// SIMATIC S7-200 project (STEP 7-Micro/WIN), CPU 224XP CN REL 02.01

ORGANIZATION_BLOCK MAIN:OB1
TITLE=程序注释
BEGIN
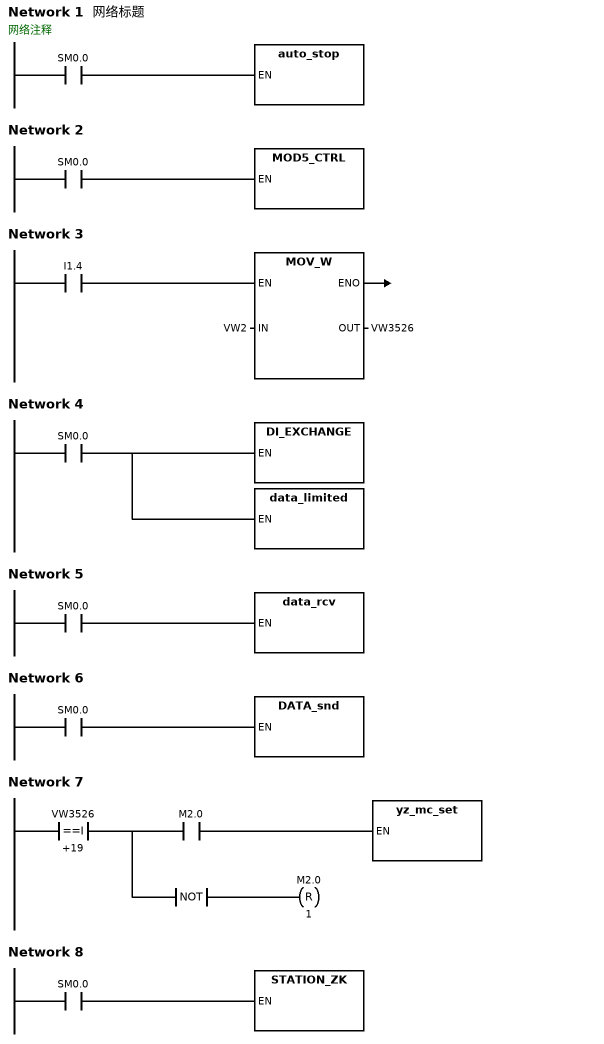
Network 1 // 网络标题
// 网络注释
LD     SM0.0
CALL   auto_stop:SBR13
Network 2
LD     SM0.0
CALL   MOD5_CTRL:SBR12
Network 3
LD     I1.4
MOVW   VW2, VW3526
Network 4
LD     SM0.0
CALL   DI_EXCHANGE:SBR4
CALL   data_limited:SBR9
Network 5
LD     SM0.0
CALL   data_rcv:SBR10
Network 6
LD     SM0.0
CALL   DATA_snd:SBR1
Network 7
LDW=   VW3526, +19
LPS
A      M2.0
CALL   yz_mc_set:SBR6
LPP
NOT
R      M2.0, 1
Network 8
LD     SM0.0
CALL   STATION_ZK:SBR2
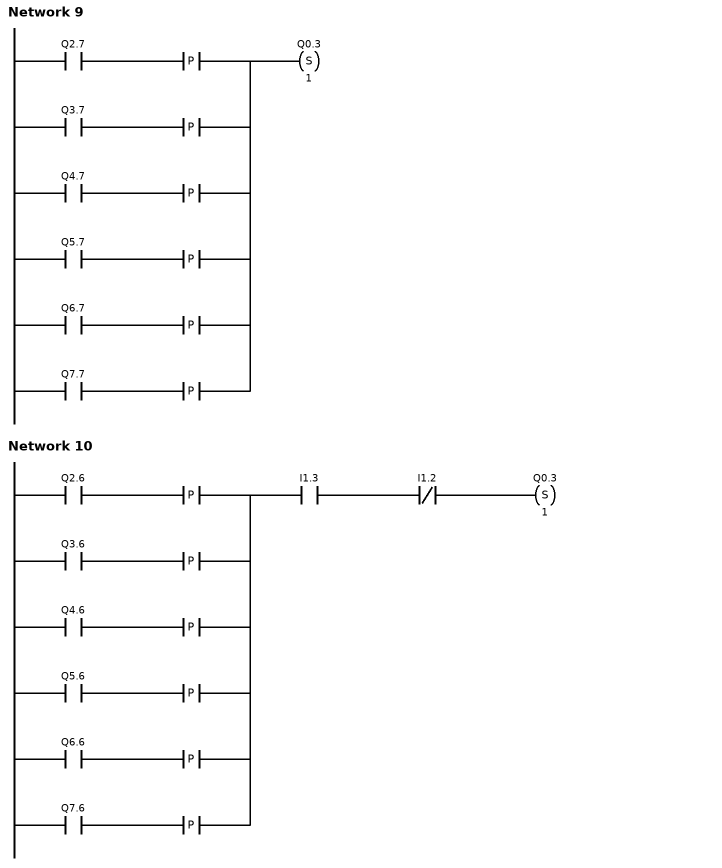
Network 9
LD     Q2.7
EU
LD     Q3.7
EU
OLD
LD     Q4.7
EU
OLD
LD     Q5.7
EU
OLD
LD     Q6.7
EU
OLD
LD     Q7.7
EU
OLD
S      Q0.3, 1
Network 10
LD     Q2.6
EU
LD     Q3.6
EU
OLD
LD     Q4.6
EU
OLD
LD     Q5.6
EU
OLD
LD     Q6.6
EU
OLD
LD     Q7.6
EU
OLD
A      I1.3
AN     I1.2
S      Q0.3, 1
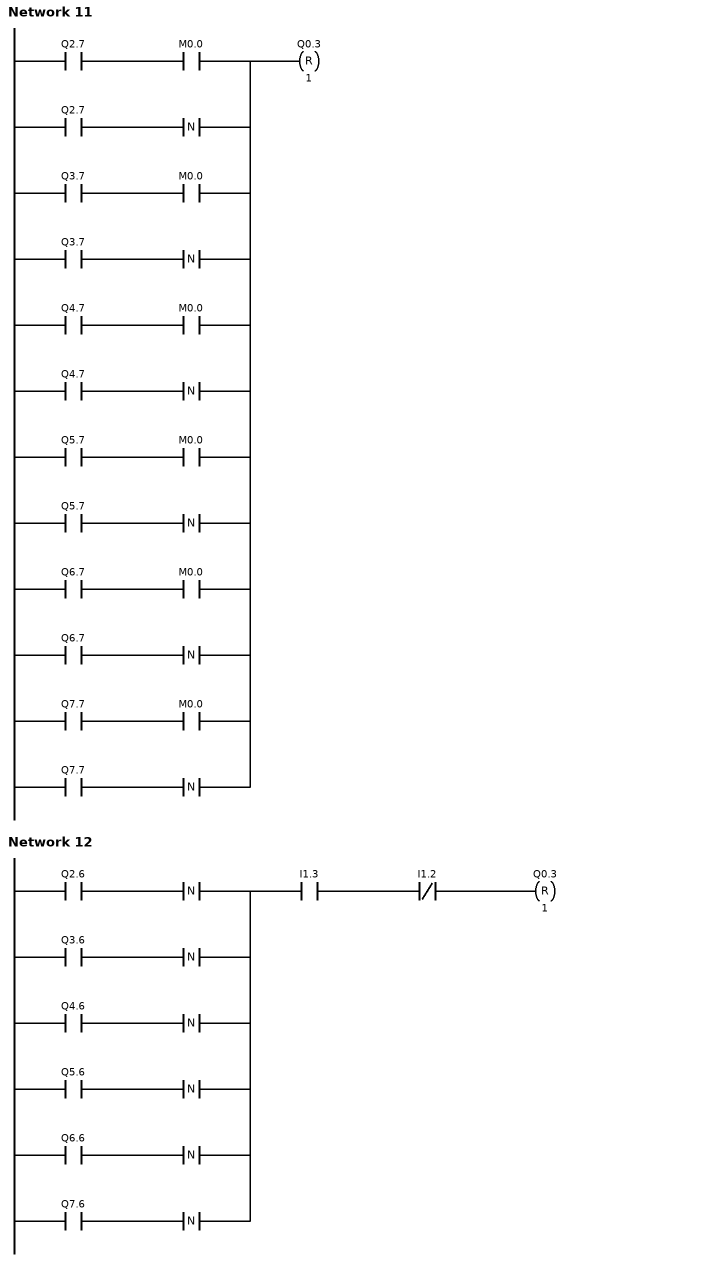
Network 11
LD     Q2.7
A      M0.0
LD     Q2.7
ED
OLD
LD     Q3.7
A      M0.0
OLD
LD     Q3.7
ED
OLD
LD     Q4.7
A      M0.0
OLD
LD     Q4.7
ED
OLD
LD     Q5.7
A      M0.0
OLD
LD     Q5.7
ED
OLD
LD     Q6.7
A      M0.0
OLD
LD     Q6.7
ED
OLD
LD     Q7.7
A      M0.0
OLD
LD     Q7.7
ED
OLD
R      Q0.3, 1
Network 12
LD     Q2.6
ED
LD     Q3.6
ED
OLD
LD     Q4.6
ED
OLD
LD     Q5.6
ED
OLD
LD     Q6.6
ED
OLD
LD     Q7.6
ED
OLD
A      I1.3
AN     I1.2
R      Q0.3, 1
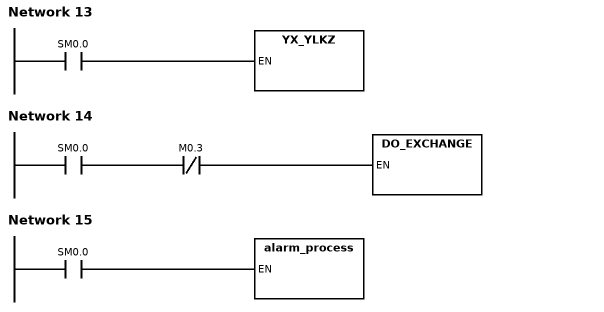
Network 13
LD     SM0.0
CALL   YX_YLKZ:SBR3
Network 14
LD     SM0.0
AN     M0.3
CALL   DO_EXCHANGE:SBR5
Network 15
LD     SM0.0
CALL   alarm_process:SBR11
END_ORGANIZATION_BLOCK

SUBROUTINE_BLOCK STATION_CONTROL:SBR0
TITLE=子程序注释
BEGIN
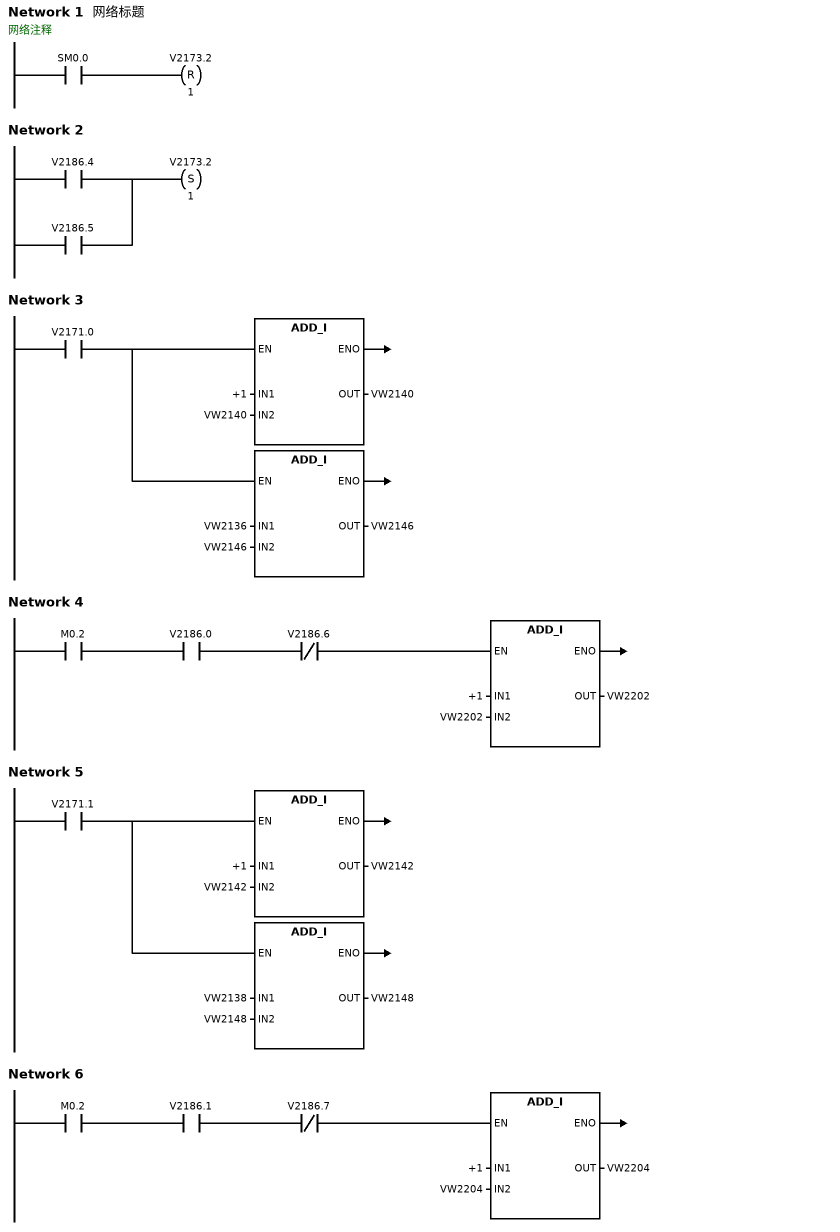
Network 1 // 网络标题
// 网络注释
LD     SM0.0
R      V2173.2, 1
Network 2
LD     V2186.4
O      V2186.5
S      V2173.2, 1
Network 3
LD     V2171.0
+I     +1, VW2140
+I     VW2136, VW2146
Network 4
LD     M0.2
A      V2186.0
AN     V2186.6
+I     +1, VW2202
Network 5
LD     V2171.1
+I     +1, VW2142
+I     VW2138, VW2148
Network 6
LD     M0.2
A      V2186.1
AN     V2186.7
+I     +1, VW2204
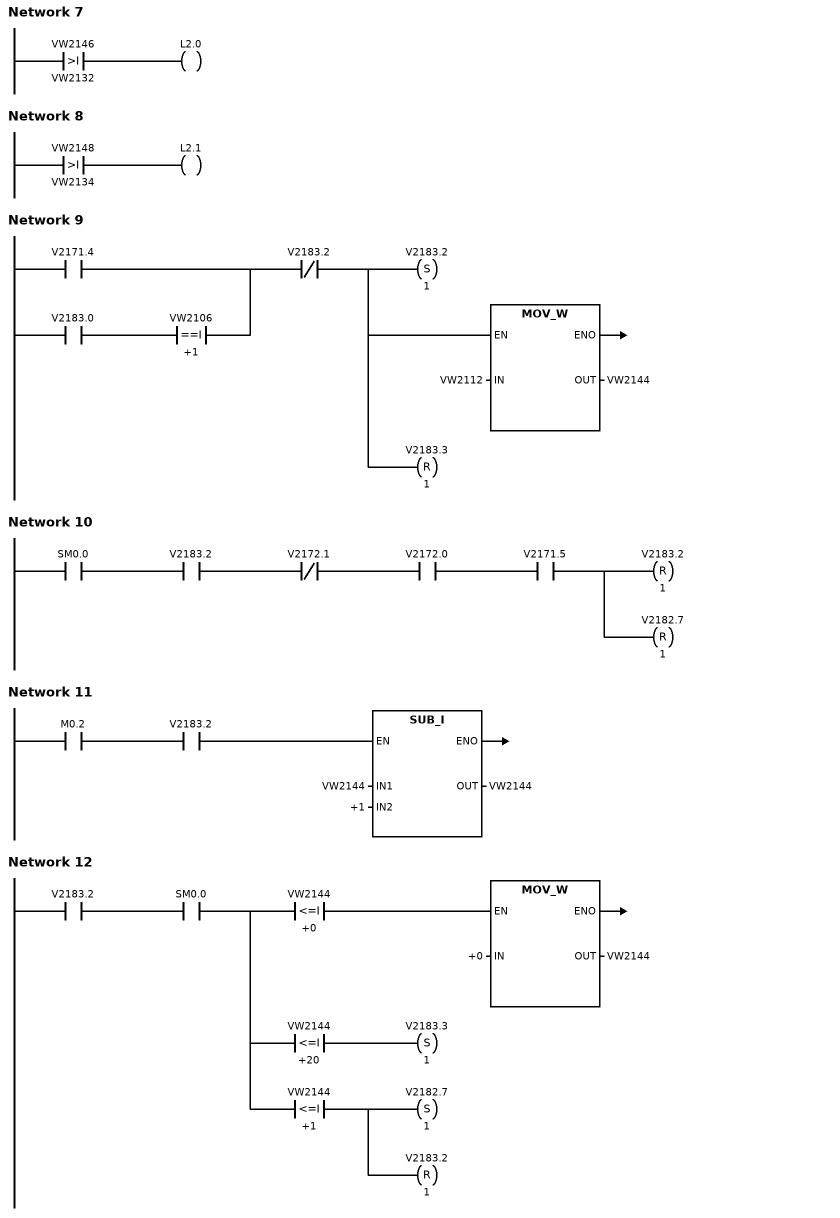
Network 7
LDW>   VW2146, VW2132
=      L2.0
Network 8
LDW>   VW2148, VW2134
=      L2.1
Network 9
LD     V2171.4
LD     V2183.0
AW=    VW2106, +1
OLD
AN     V2183.2
S      V2183.2, 1
MOVW   VW2112, VW2144
R      V2183.3, 1
Network 10
LD     SM0.0
A      V2183.2
AN     V2172.1
A      V2172.0
A      V2171.5
R      V2183.2, 1
R      V2182.7, 1
Network 11
LD     M0.2
A      V2183.2
-I     +1, VW2144
Network 12
LD     V2183.2
A      SM0.0
LPS
AW<=   VW2144, +0
MOVW   +0, VW2144
LRD
AW<=   VW2144, +20
S      V2183.3, 1
LPP
AW<=   VW2144, +1
S      V2182.7, 1
R      V2183.2, 1
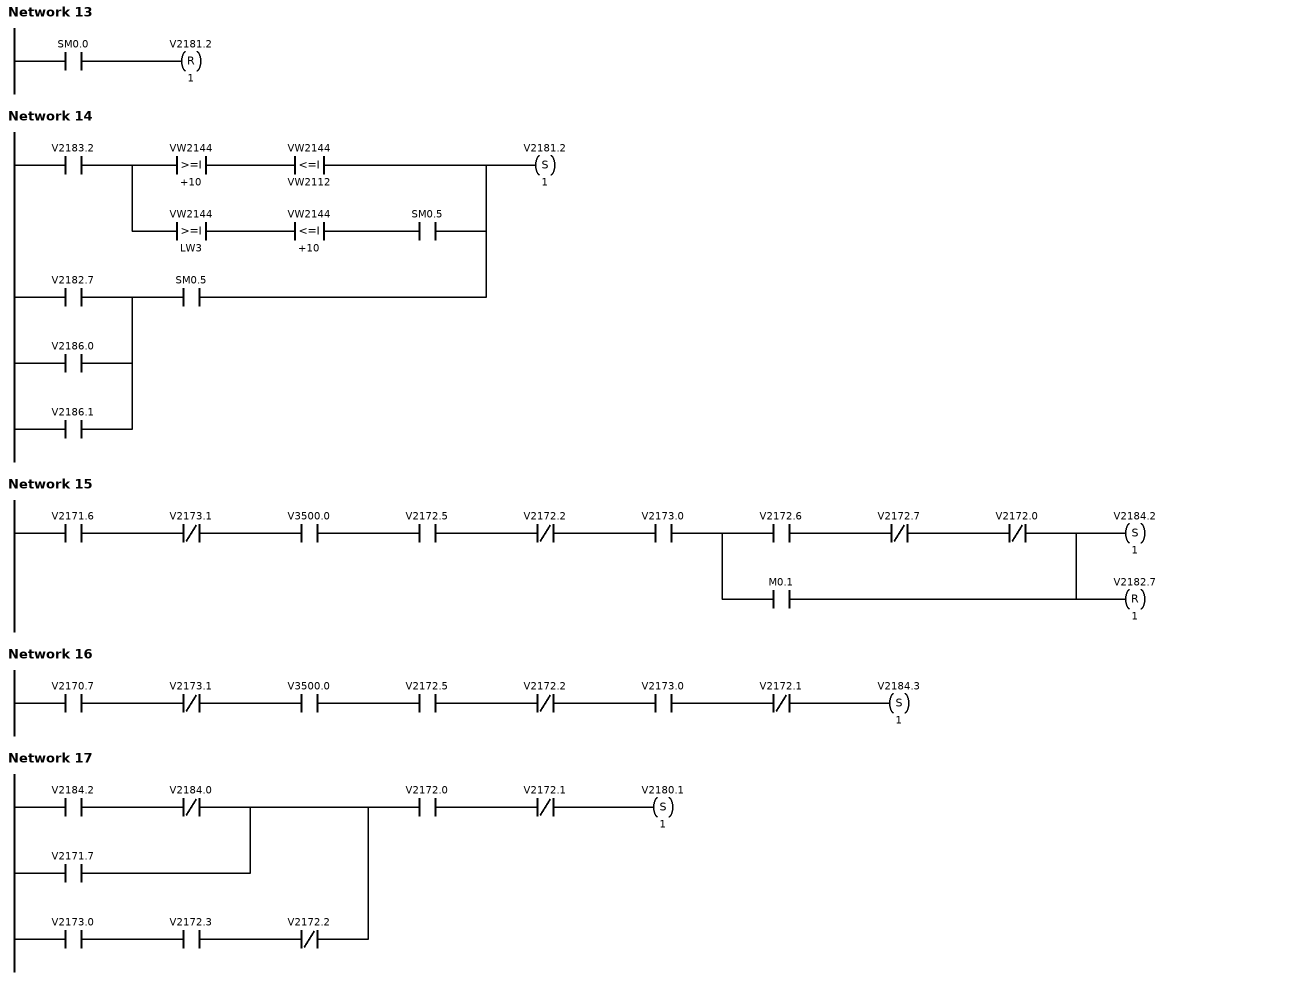
Network 13
LD     SM0.0
R      V2181.2, 1
Network 14
LD     V2183.2
LDW>=  VW2144, +10
AW<=   VW2144, VW2112
LDW>=  VW2144, LW3
AW<=   VW2144, +10
A      SM0.5
OLD
ALD
LD     V2182.7
O      V2186.0
O      V2186.1
A      SM0.5
OLD
S      V2181.2, 1
Network 15
LD     V2171.6
AN     V2173.1
A      V3500.0
A      V2172.5
AN     V2172.2
A      V2173.0
LD     V2172.6
AN     V2172.7
AN     V2172.0
O      M0.1
ALD
S      V2184.2, 1
R      V2182.7, 1
Network 16
LD     V2170.7
AN     V2173.1
A      V3500.0
A      V2172.5
AN     V2172.2
A      V2173.0
AN     V2172.1
S      V2184.3, 1
Network 17
LD     V2184.2
AN     V2184.0
O      V2171.7
LD     V2173.0
A      V2172.3
AN     V2172.2
OLD
A      V2172.0
AN     V2172.1
S      V2180.1, 1
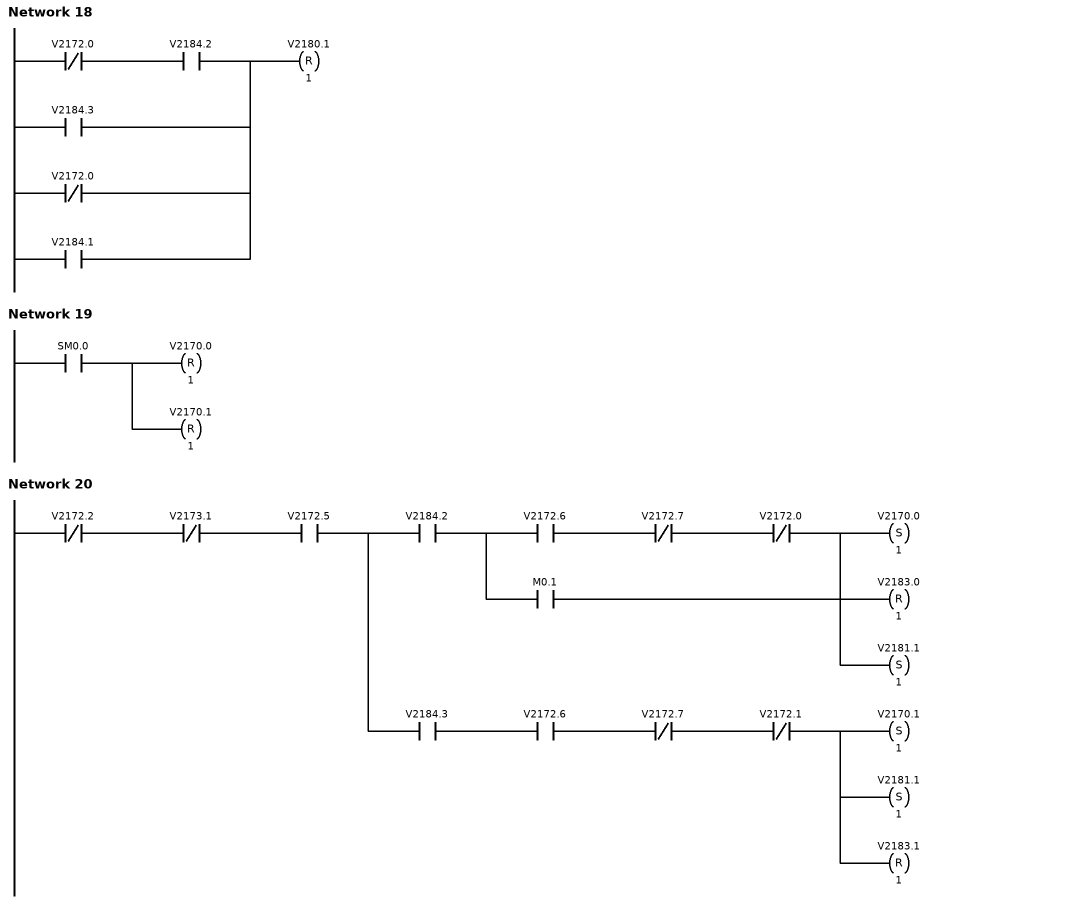
Network 18
LDN    V2172.0
A      V2184.2
O      V2184.3
ON     V2172.0
O      V2184.1
R      V2180.1, 1
Network 19
LD     SM0.0
R      V2170.0, 1
R      V2170.1, 1
Network 20
LDN    V2172.2
AN     V2173.1
A      V2172.5
LPS
A      V2184.2
LD     V2172.6
AN     V2172.7
AN     V2172.0
O      M0.1
ALD
S      V2170.0, 1
R      V2183.0, 1
S      V2181.1, 1
LPP
A      V2184.3
A      V2172.6
AN     V2172.7
AN     V2172.1
S      V2170.1, 1
S      V2181.1, 1
R      V2183.1, 1
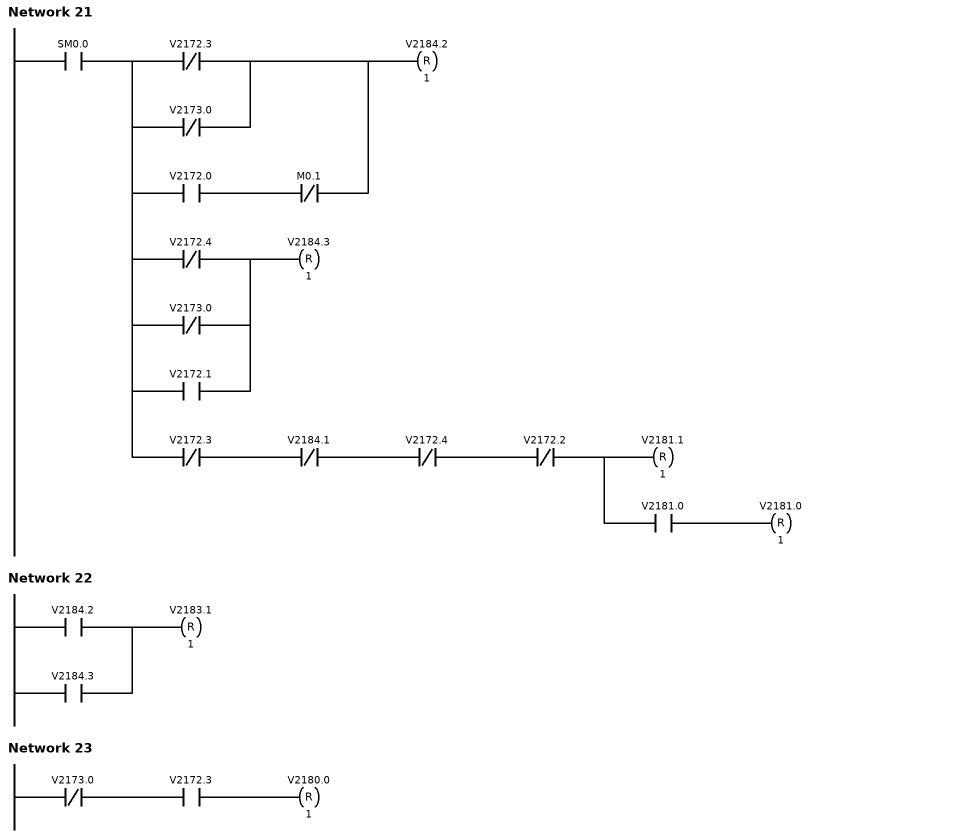
Network 21
LD     SM0.0
LPS
LDN    V2172.3
ON     V2173.0
LD     V2172.0
AN     M0.1
OLD
ALD
R      V2184.2, 1
LRD
LDN    V2172.4
ON     V2173.0
O      V2172.1
ALD
R      V2184.3, 1
LPP
AN     V2172.3
AN     V2184.1
AN     V2172.4
AN     V2172.2
R      V2181.1, 1
A      V2181.0
R      V2181.0, 1
Network 22
LD     V2184.2
O      V2184.3
R      V2183.1, 1
Network 23
LDN    V2173.0
A      V2172.3
R      V2180.0, 1
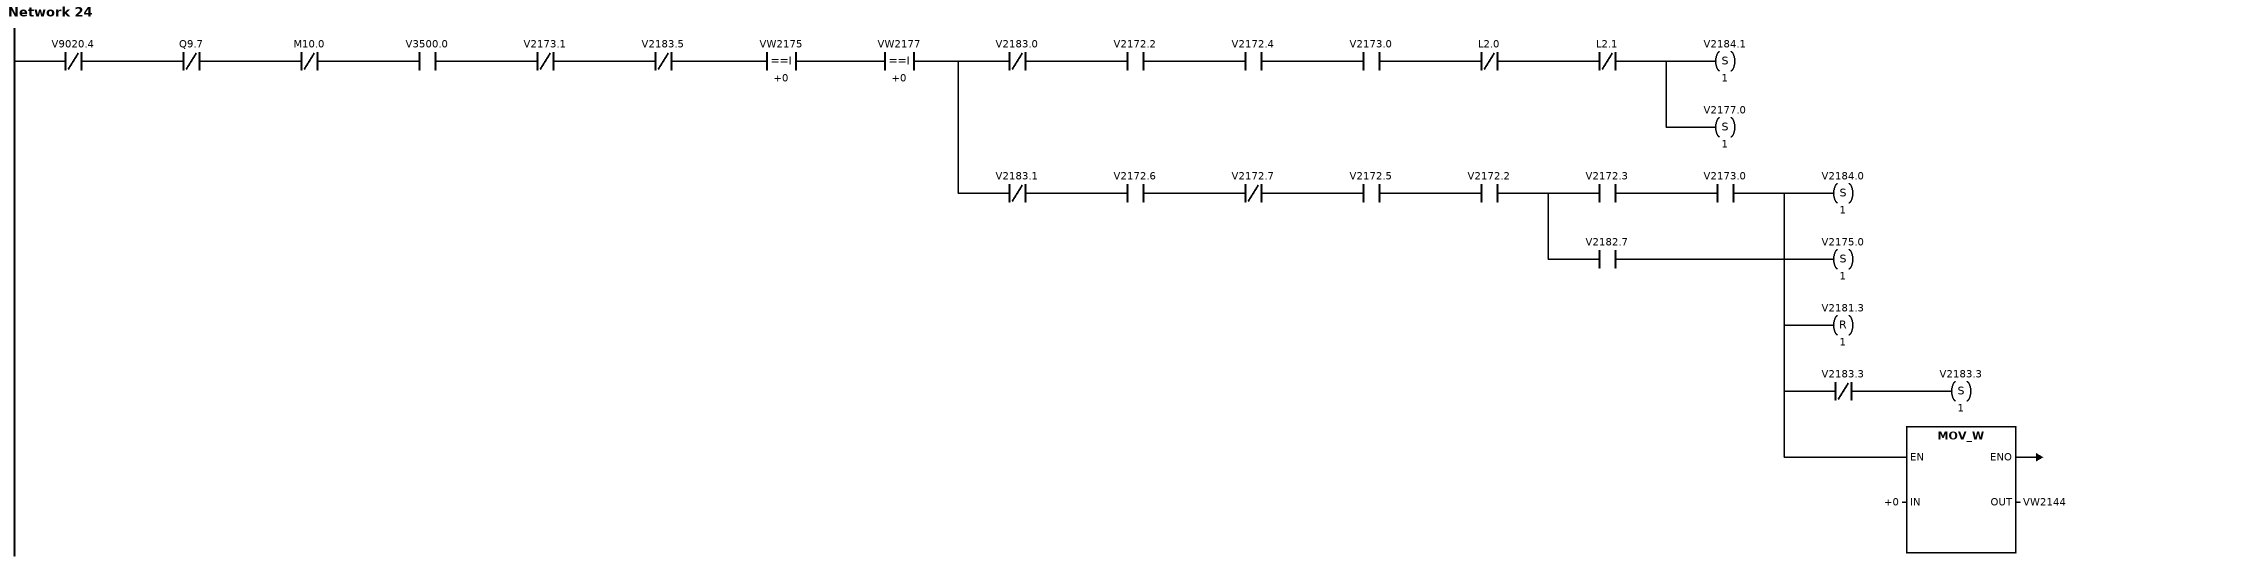
Network 24
LDN    V9020.4
AN     Q9.7
AN     M10.0
A      V3500.0
AN     V2173.1
AN     V2183.5
AW=    VW2175, +0
AW=    VW2177, +0
LPS
AN     V2183.0
A      V2172.2
A      V2172.4
A      V2173.0
AN     L2.0
AN     L2.1
S      V2184.1, 1
S      V2177.0, 1
LPP
AN     V2183.1
A      V2172.6
AN     V2172.7
A      V2172.5
A      V2172.2
LD     V2172.3
A      V2173.0
O      V2182.7
ALD
LPS
S      V2184.0, 1
S      V2175.0, 1
R      V2181.3, 1
AN     V2183.3
S      V2183.3, 1
LPP
MOVW   +0, VW2144
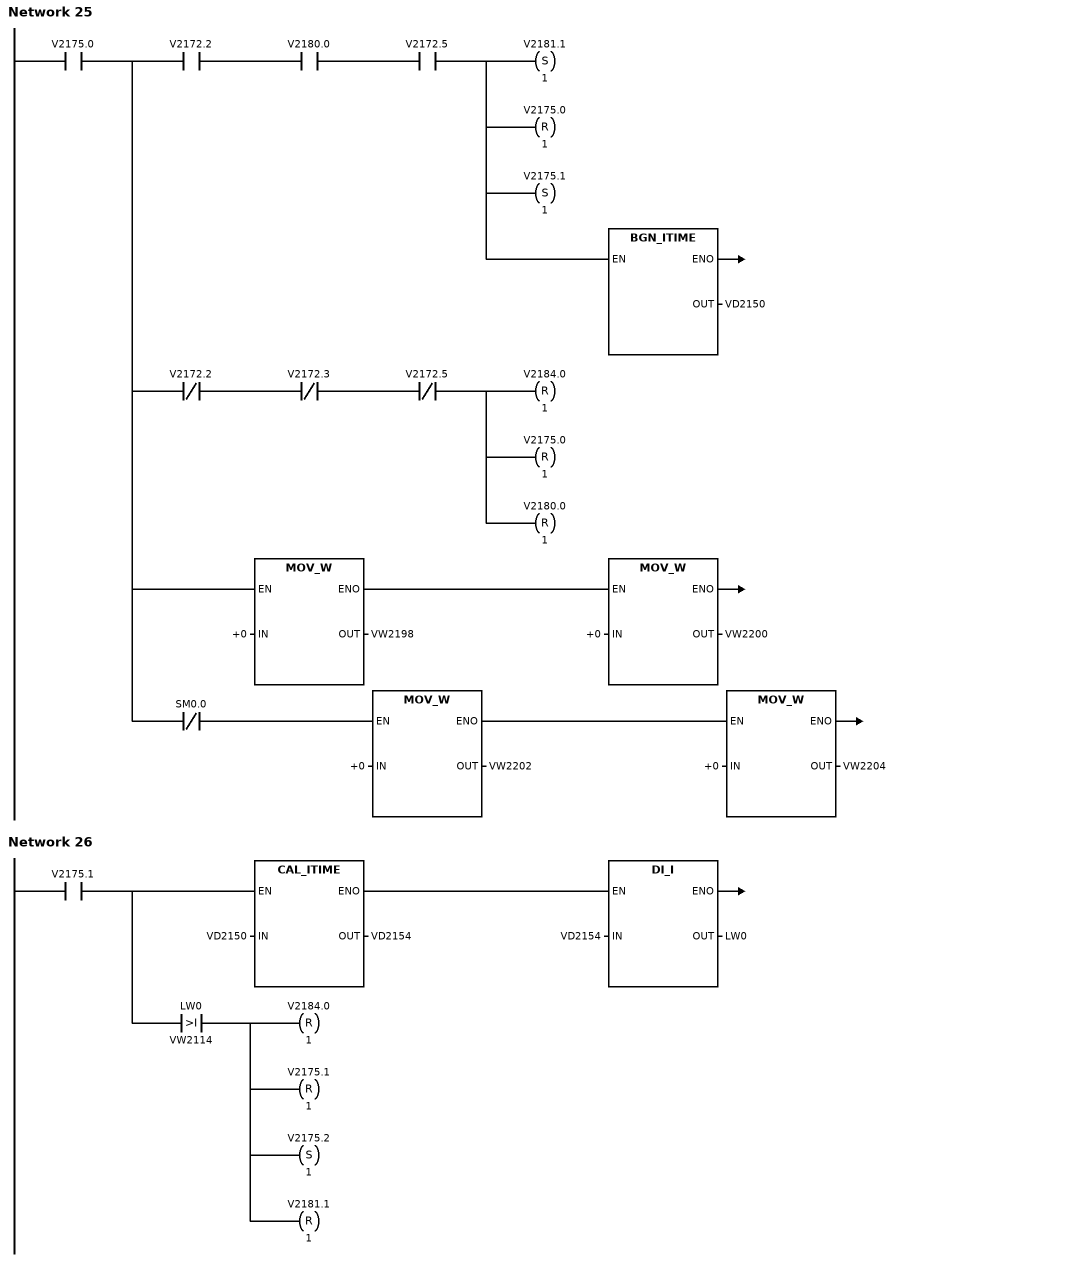
Network 25
LD     V2175.0
LPS
A      V2172.2
A      V2180.0
A      V2172.5
S      V2181.1, 1
R      V2175.0, 1
S      V2175.1, 1
BITIM  VD2150
LRD
AN     V2172.2
AN     V2172.3
AN     V2172.5
R      V2184.0, 1
R      V2175.0, 1
R      V2180.0, 1
LPP
LPS
MOVW   +0, VW2198
AENO
MOVW   +0, VW2200
LPP
AN     SM0.0
MOVW   +0, VW2202
AENO
MOVW   +0, VW2204
Network 26
LD     V2175.1
LPS
CITIM  VD2150, VD2154
AENO
DTI    VD2154, LW0
LPP
AW>    LW0, VW2114
R      V2184.0, 1
R      V2175.1, 1
S      V2175.2, 1
R      V2181.1, 1
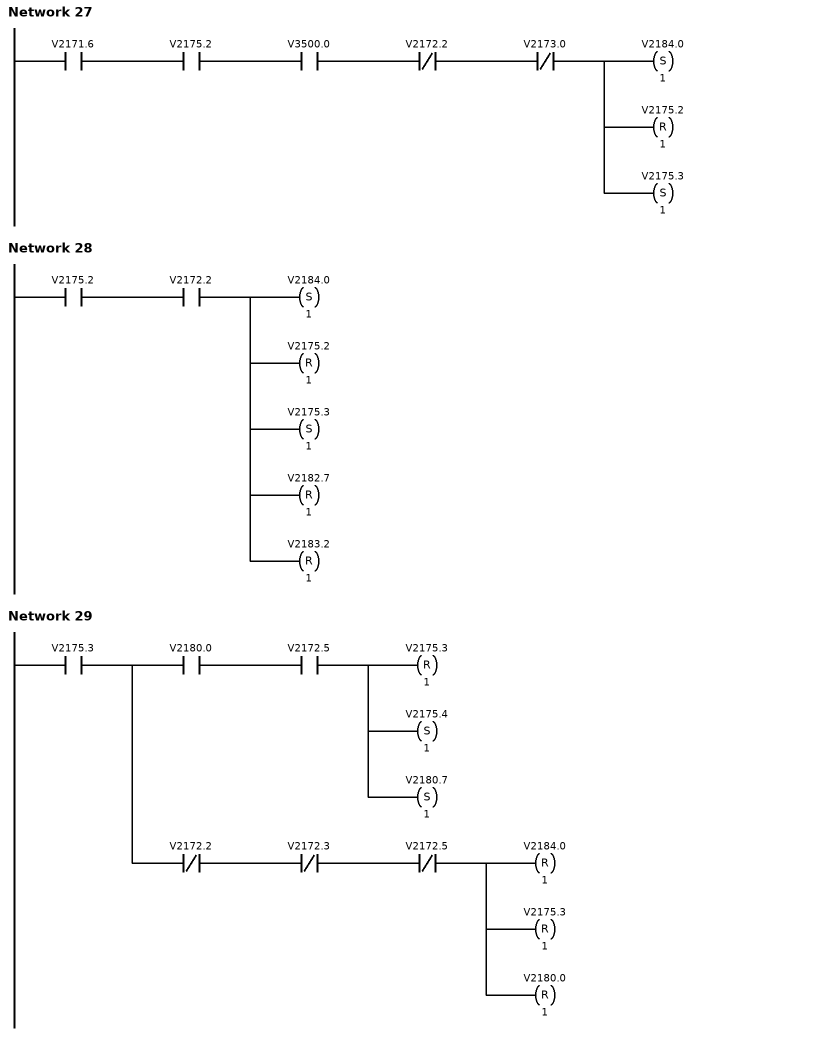
Network 27
LD     V2171.6
A      V2175.2
A      V3500.0
AN     V2172.2
AN     V2173.0
S      V2184.0, 1
R      V2175.2, 1
S      V2175.3, 1
Network 28
LD     V2175.2
A      V2172.2
S      V2184.0, 1
R      V2175.2, 1
S      V2175.3, 1
R      V2182.7, 1
R      V2183.2, 1
Network 29
LD     V2175.3
LPS
A      V2180.0
A      V2172.5
R      V2175.3, 1
S      V2175.4, 1
S      V2180.7, 1
LPP
AN     V2172.2
AN     V2172.3
AN     V2172.5
R      V2184.0, 1
R      V2175.3, 1
R      V2180.0, 1
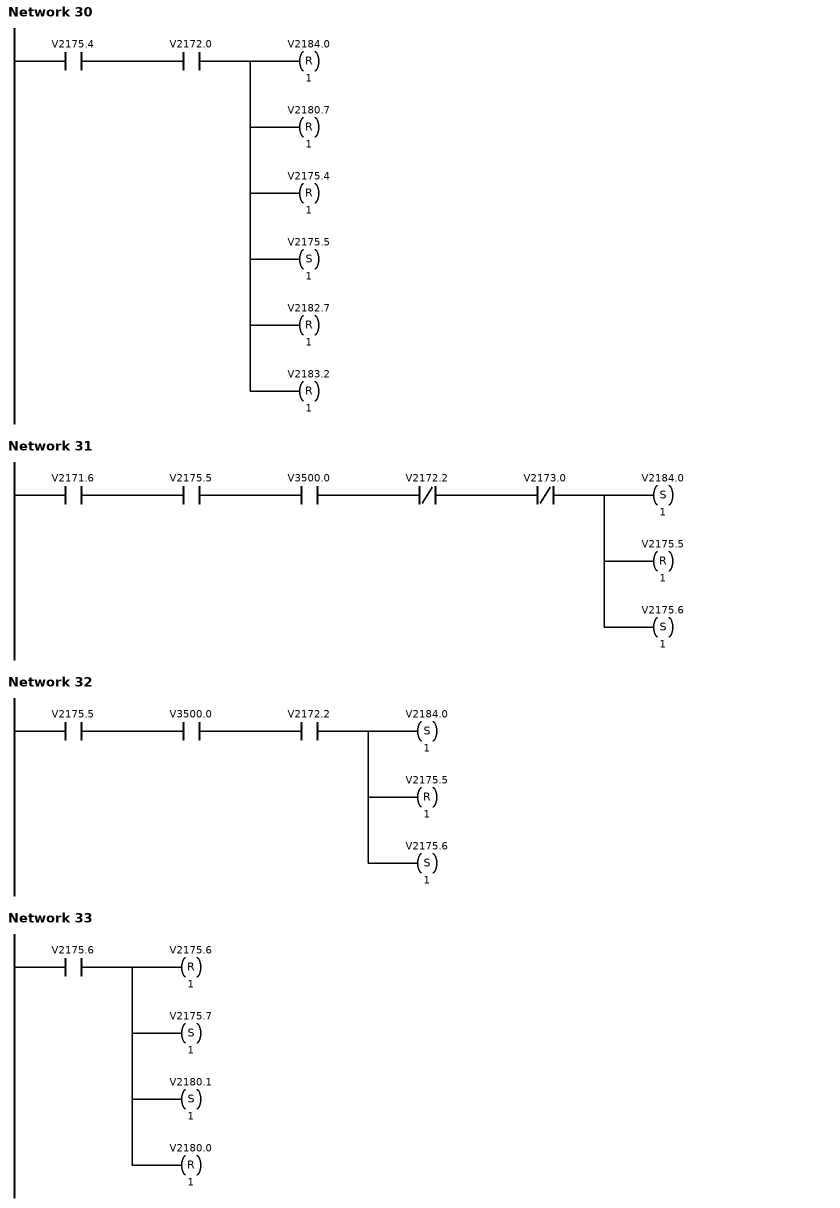
Network 30
LD     V2175.4
A      V2172.0
R      V2184.0, 1
R      V2180.7, 1
R      V2175.4, 1
S      V2175.5, 1
R      V2182.7, 1
R      V2183.2, 1
Network 31
LD     V2171.6
A      V2175.5
A      V3500.0
AN     V2172.2
AN     V2173.0
S      V2184.0, 1
R      V2175.5, 1
S      V2175.6, 1
Network 32
LD     V2175.5
A      V3500.0
A      V2172.2
S      V2184.0, 1
R      V2175.5, 1
S      V2175.6, 1
Network 33
LD     V2175.6
R      V2175.6, 1
S      V2175.7, 1
S      V2180.1, 1
R      V2180.0, 1
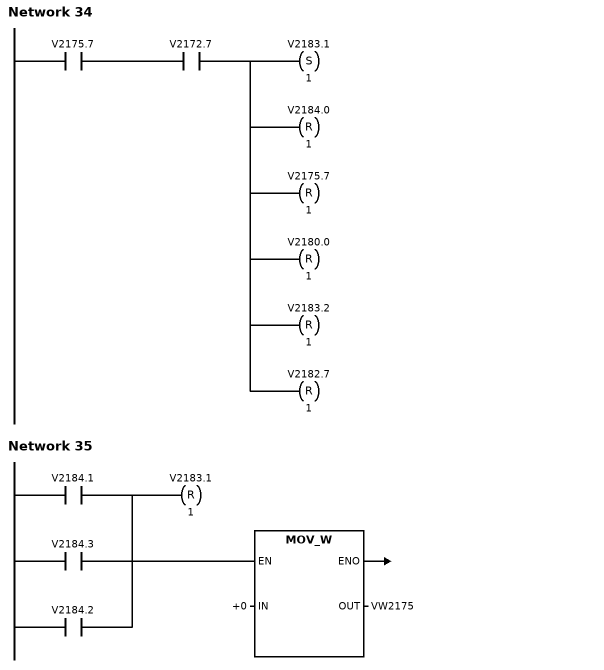
Network 34
LD     V2175.7
A      V2172.7
S      V2183.1, 1
R      V2184.0, 1
R      V2175.7, 1
R      V2180.0, 1
R      V2183.2, 1
R      V2182.7, 1
Network 35
LD     V2184.1
O      V2184.3
O      V2184.2
R      V2183.1, 1
MOVW   +0, VW2175
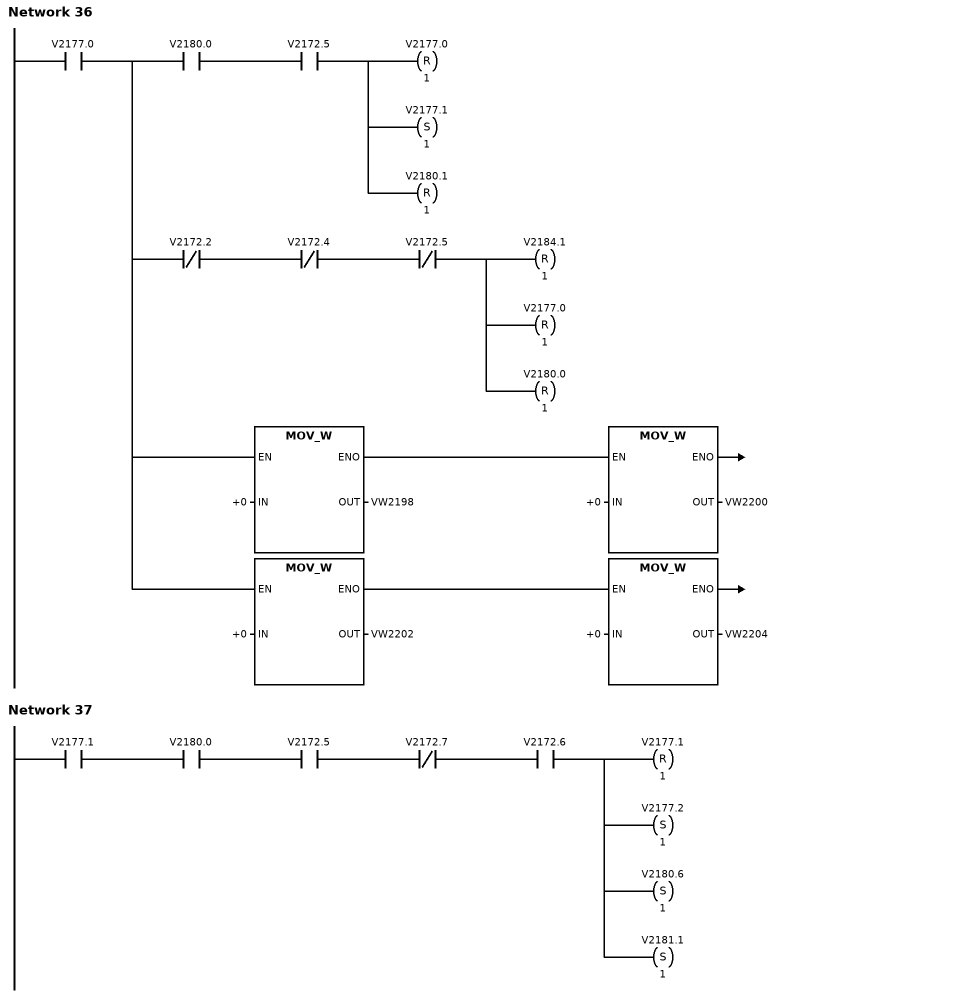
Network 36
LD     V2177.0
LPS
A      V2180.0
A      V2172.5
R      V2177.0, 1
S      V2177.1, 1
R      V2180.1, 1
LRD
AN     V2172.2
AN     V2172.4
AN     V2172.5
R      V2184.1, 1
R      V2177.0, 1
R      V2180.0, 1
LPP
LPS
MOVW   +0, VW2198
AENO
MOVW   +0, VW2200
LPP
MOVW   +0, VW2202
AENO
MOVW   +0, VW2204
Network 37
LD     V2177.1
A      V2180.0
A      V2172.5
AN     V2172.7
A      V2172.6
R      V2177.1, 1
S      V2177.2, 1
S      V2180.6, 1
S      V2181.1, 1
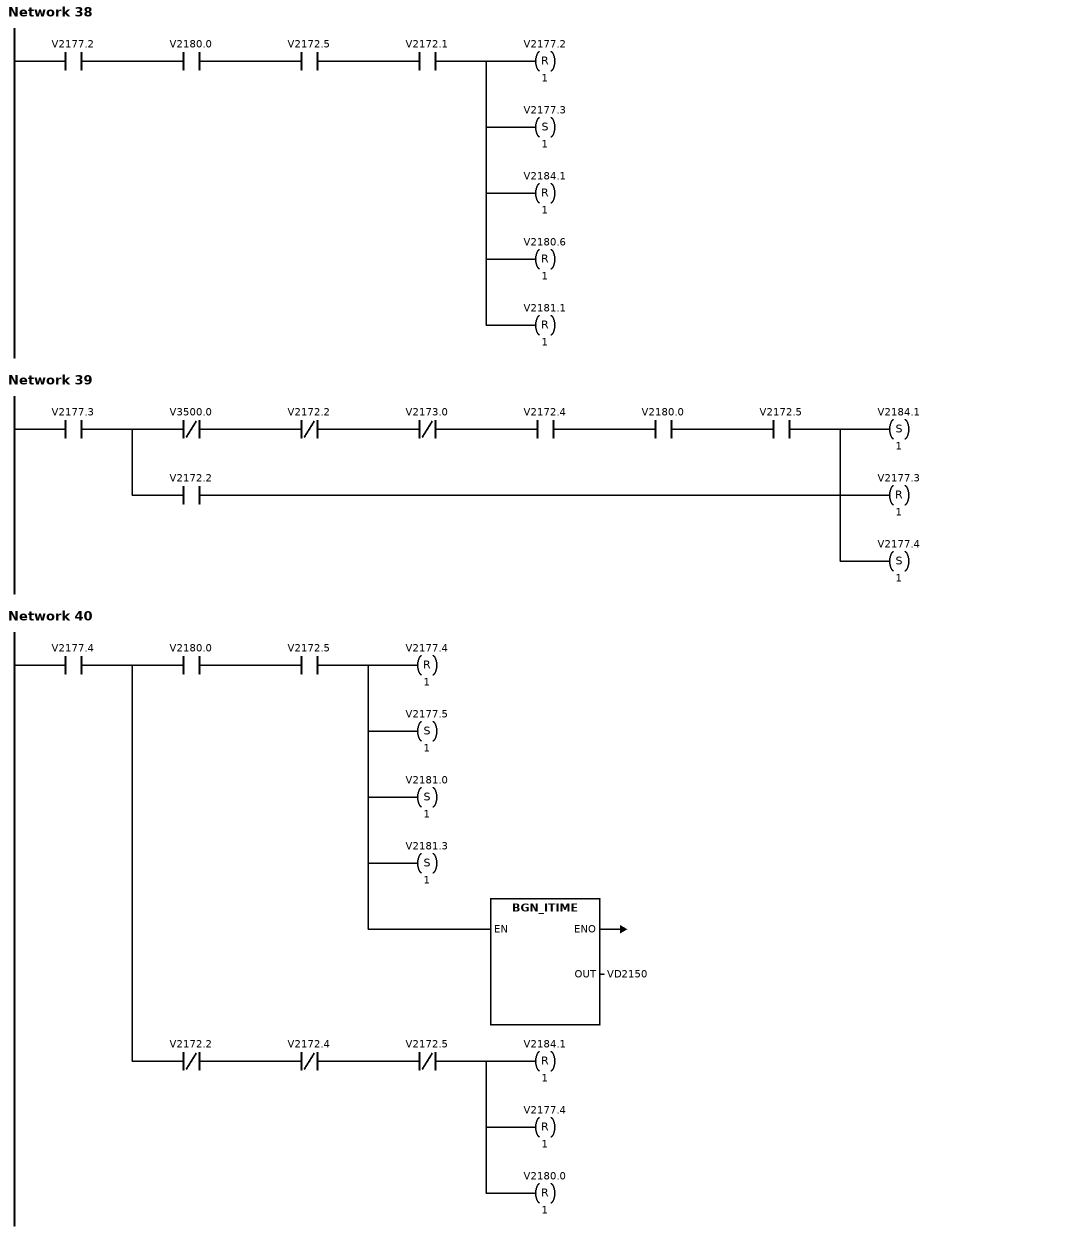
Network 38
LD     V2177.2
A      V2180.0
A      V2172.5
A      V2172.1
R      V2177.2, 1
S      V2177.3, 1
R      V2184.1, 1
R      V2180.6, 1
R      V2181.1, 1
Network 39
LD     V2177.3
LDN    V3500.0
AN     V2172.2
AN     V2173.0
A      V2172.4
A      V2180.0
A      V2172.5
O      V2172.2
ALD
S      V2184.1, 1
R      V2177.3, 1
S      V2177.4, 1
Network 40
LD     V2177.4
LPS
A      V2180.0
A      V2172.5
R      V2177.4, 1
S      V2177.5, 1
S      V2181.0, 1
S      V2181.3, 1
BITIM  VD2150
LPP
AN     V2172.2
AN     V2172.4
AN     V2172.5
R      V2184.1, 1
R      V2177.4, 1
R      V2180.0, 1
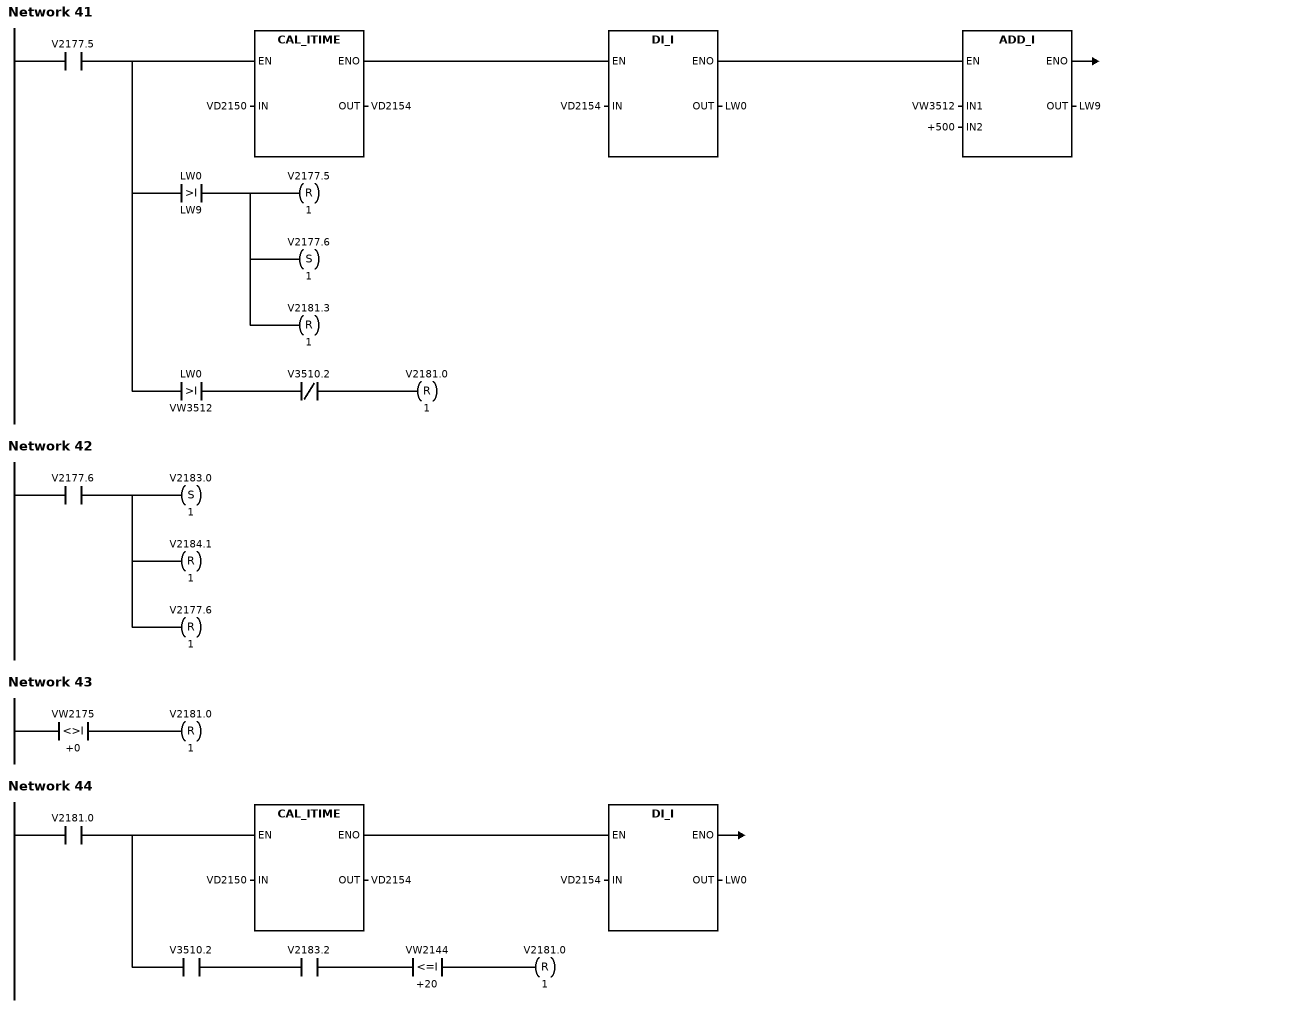
Network 41
LD     V2177.5
LPS
CITIM  VD2150, VD2154
AENO
DTI    VD2154, LW0
AENO
MOVW   VW3512, LW9
+I     +500, LW9
LRD
AW>    LW0, LW9
R      V2177.5, 1
S      V2177.6, 1
R      V2181.3, 1
LPP
AW>    LW0, VW3512
AN     V3510.2
R      V2181.0, 1
Network 42
LD     V2177.6
S      V2183.0, 1
R      V2184.1, 1
R      V2177.6, 1
Network 43
LDW<>  VW2175, +0
R      V2181.0, 1
Network 44
LD     V2181.0
LPS
CITIM  VD2150, VD2154
AENO
DTI    VD2154, LW0
LPP
A      V3510.2
A      V2183.2
AW<=   VW2144, +20
R      V2181.0, 1
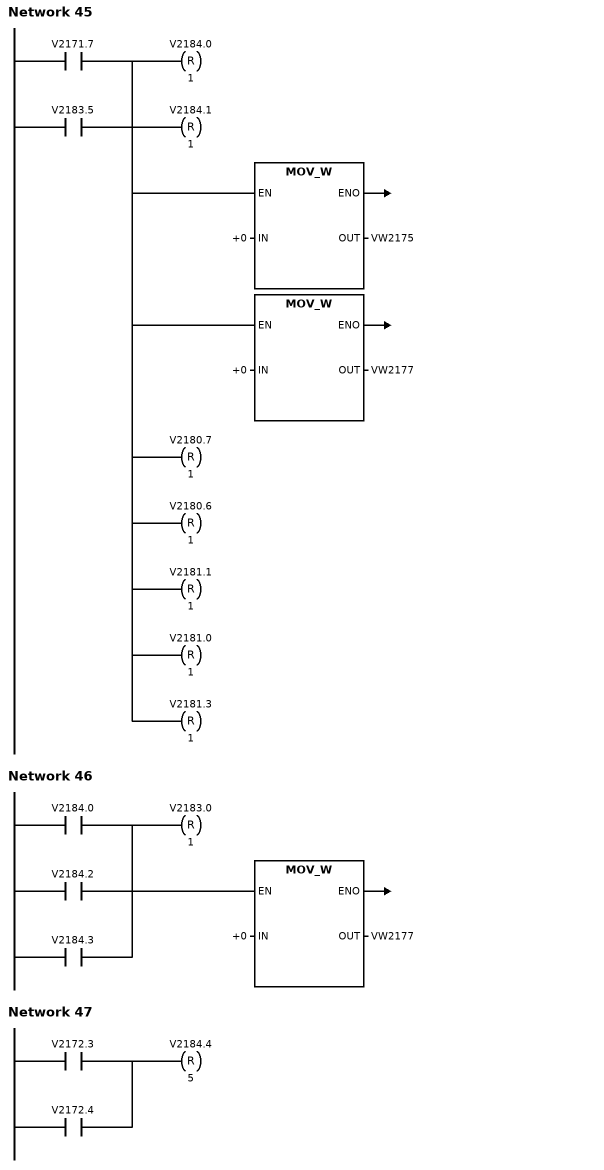
Network 45
LD     V2171.7
O      V2183.5
R      V2184.0, 1
R      V2184.1, 1
MOVW   +0, VW2175
MOVW   +0, VW2177
R      V2180.7, 1
R      V2180.6, 1
R      V2181.1, 1
R      V2181.0, 1
R      V2181.3, 1
Network 46
LD     V2184.0
O      V2184.2
O      V2184.3
R      V2183.0, 1
MOVW   +0, VW2177
Network 47
LD     V2172.3
O      V2172.4
R      V2184.4, 5
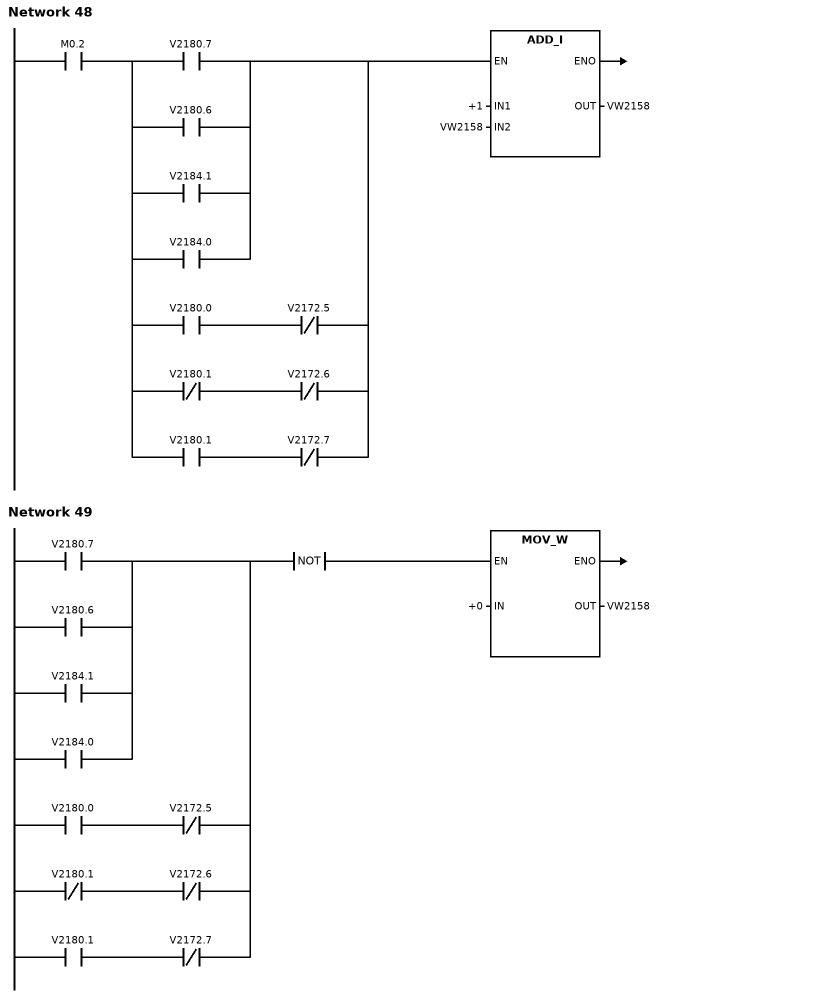
Network 48
LD     M0.2
LD     V2180.7
O      V2180.6
O      V2184.1
O      V2184.0
LD     V2180.0
AN     V2172.5
OLD
LDN    V2180.1
AN     V2172.6
OLD
LD     V2180.1
AN     V2172.7
OLD
ALD
+I     +1, VW2158
Network 49
LD     V2180.7
O      V2180.6
O      V2184.1
O      V2184.0
LD     V2180.0
AN     V2172.5
OLD
LDN    V2180.1
AN     V2172.6
OLD
LD     V2180.1
AN     V2172.7
OLD
NOT
MOVW   +0, VW2158
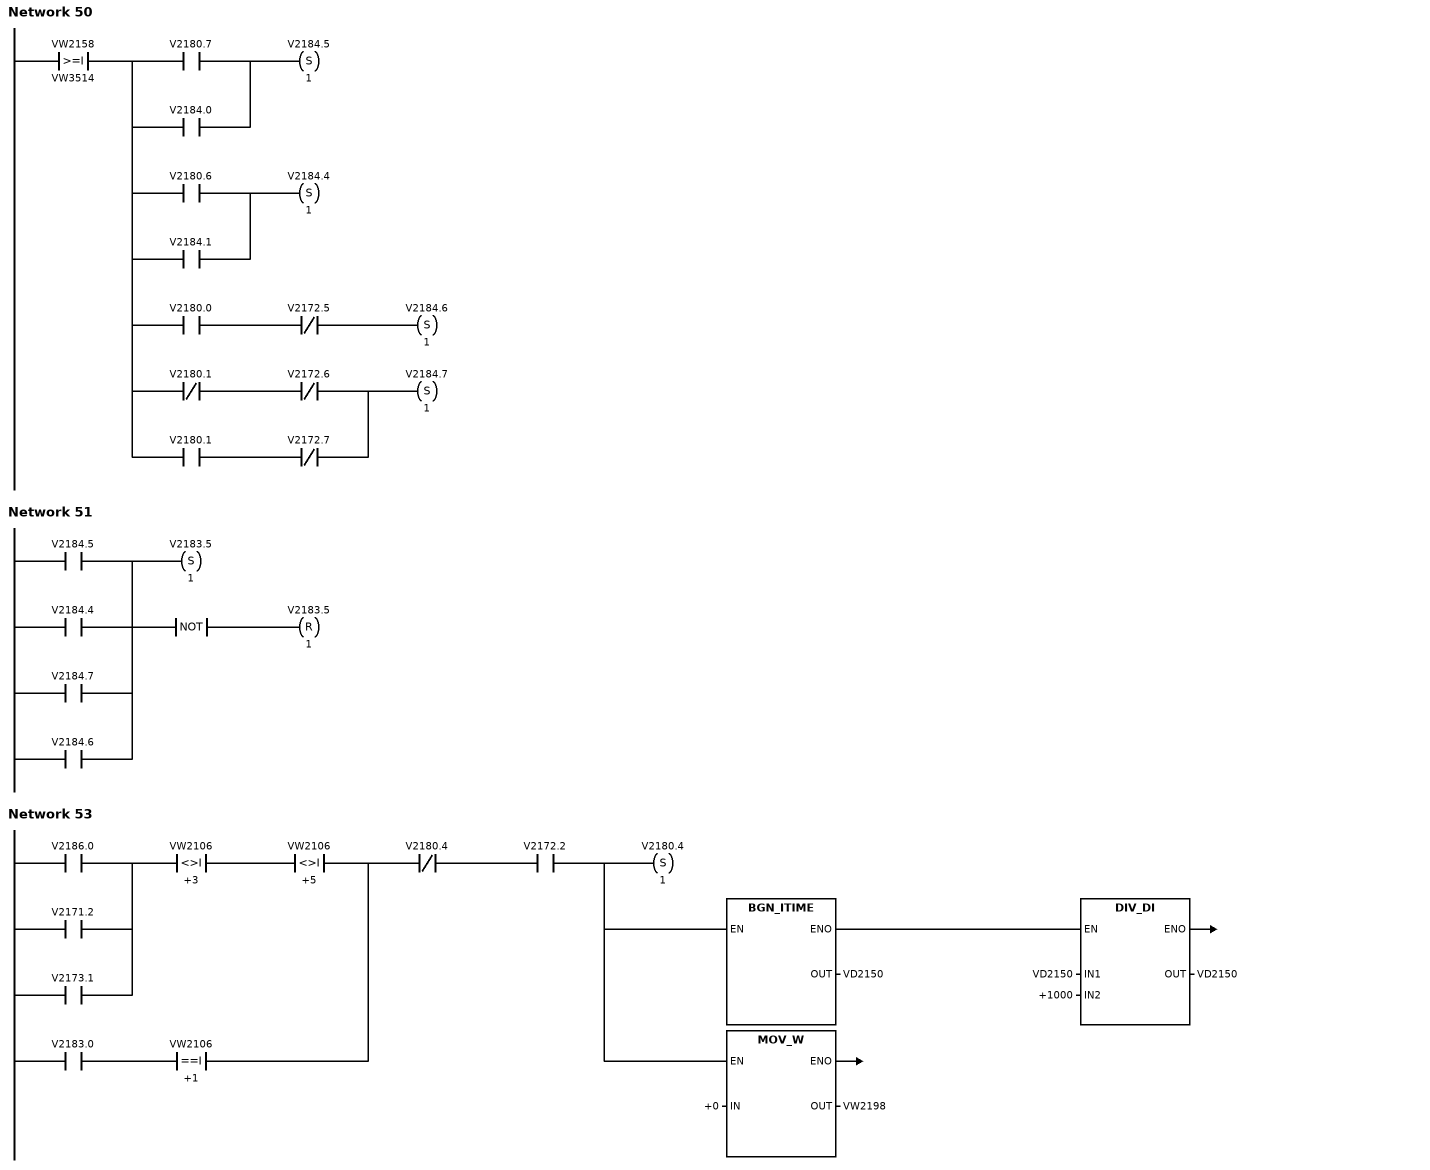
Network 50
LDW>=  VW2158, VW3514
LPS
LD     V2180.7
O      V2184.0
ALD
S      V2184.5, 1
LRD
LD     V2180.6
O      V2184.1
ALD
S      V2184.4, 1
LRD
A      V2180.0
AN     V2172.5
S      V2184.6, 1
LPP
LDN    V2180.1
AN     V2172.6
LD     V2180.1
AN     V2172.7
OLD
ALD
S      V2184.7, 1
Network 51
LD     V2184.5
O      V2184.4
O      V2184.7
O      V2184.6
S      V2183.5, 1
NOT
R      V2183.5, 1
Network 53
LD     V2186.0
O      V2171.2
O      V2173.1
AW<>   VW2106, +3
AW<>   VW2106, +5
LD     V2183.0
AW=    VW2106, +1
OLD
AN     V2180.4
A      V2172.2
LPS
S      V2180.4, 1
BITIM  VD2150
AENO
/D     +1000, VD2150
LPP
MOVW   +0, VW2198
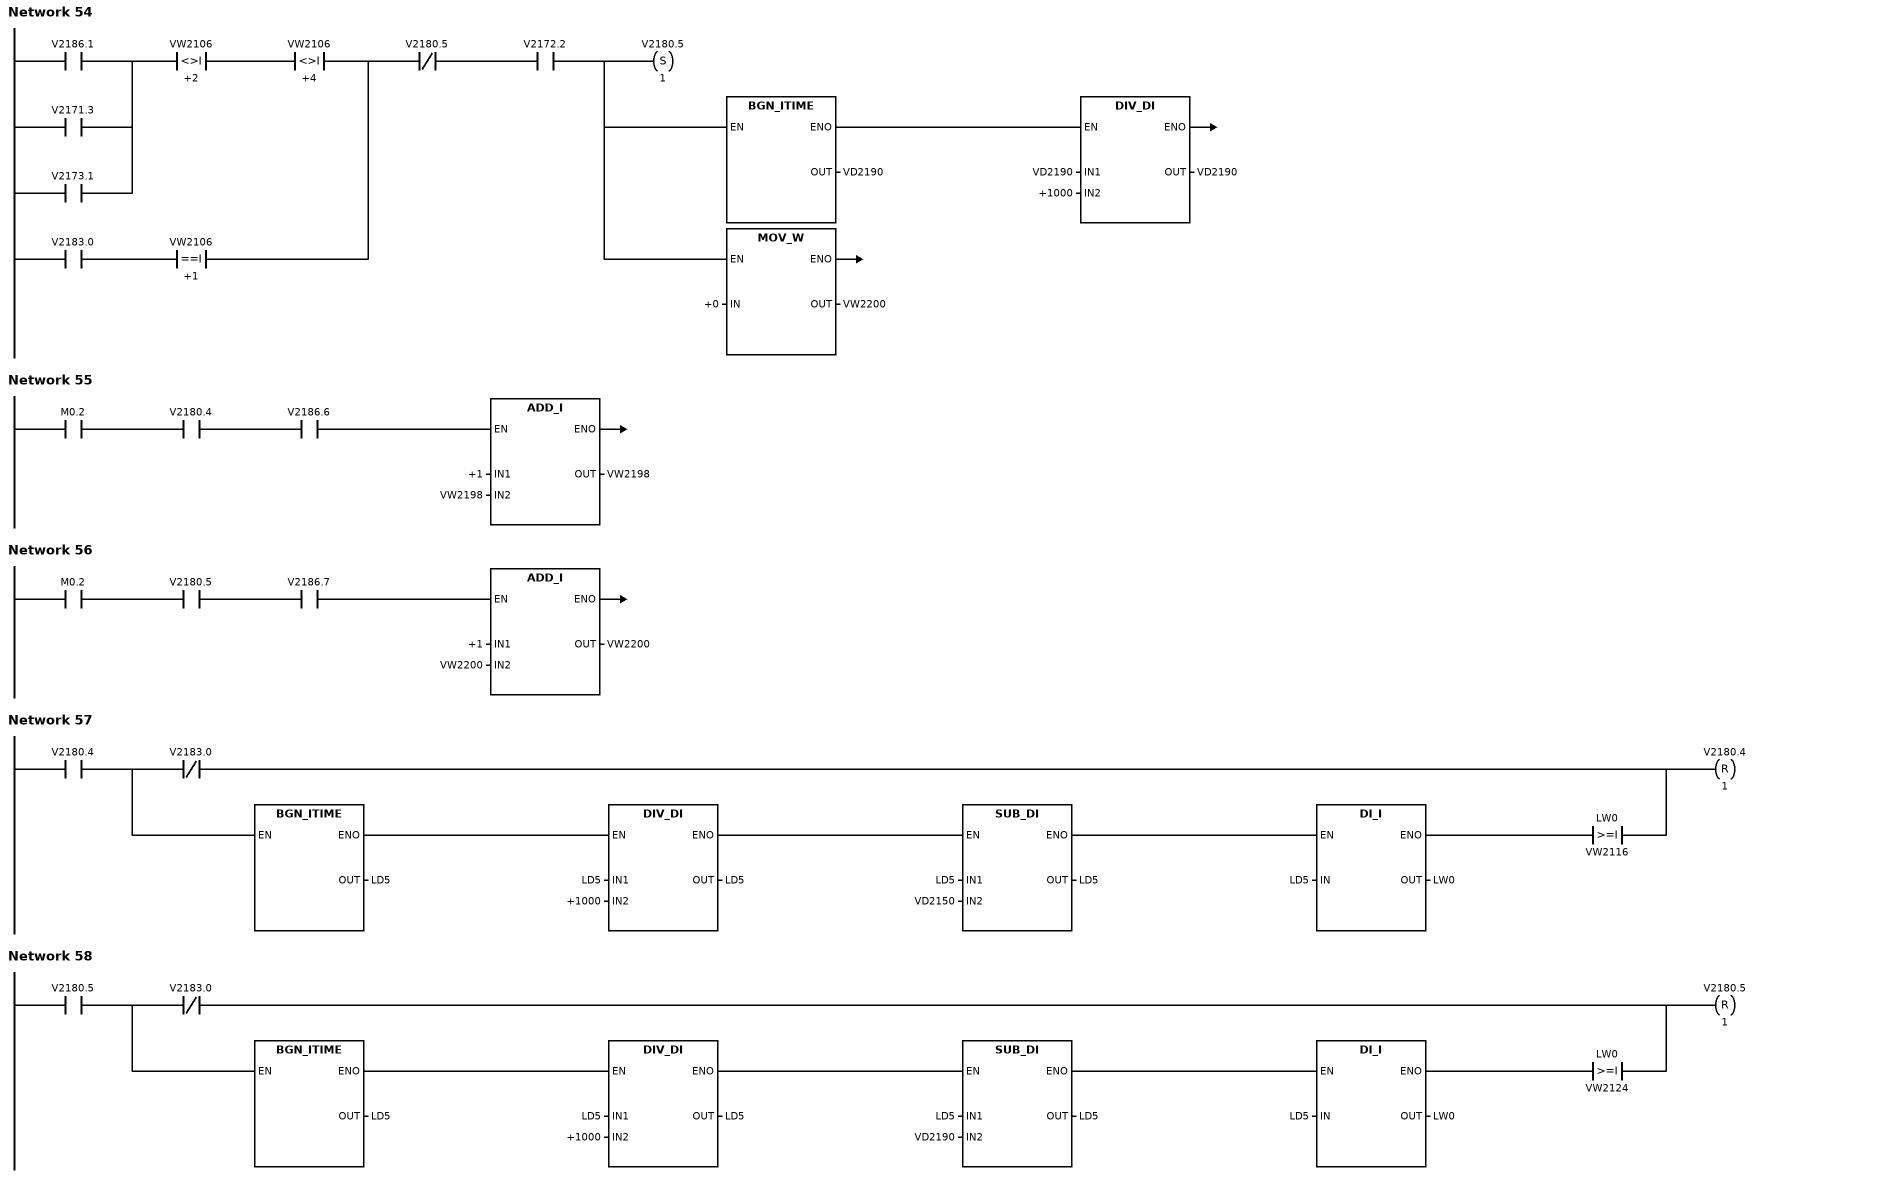
Network 54
LD     V2186.1
O      V2171.3
O      V2173.1
AW<>   VW2106, +2
AW<>   VW2106, +4
LD     V2183.0
AW=    VW2106, +1
OLD
AN     V2180.5
A      V2172.2
LPS
S      V2180.5, 1
BITIM  VD2190
AENO
/D     +1000, VD2190
LPP
MOVW   +0, VW2200
Network 55
LD     M0.2
A      V2180.4
A      V2186.6
+I     +1, VW2198
Network 56
LD     M0.2
A      V2180.5
A      V2186.7
+I     +1, VW2200
Network 57
LD     V2180.4
LPS
AN     V2183.0
=      L63.7
LPP
BITIM  LD5
AENO
/D     +1000, LD5
AENO
-D     VD2150, LD5
AENO
DTI    LD5, LW0
AENO
AW>=   LW0, VW2116
O      L63.7
R      V2180.4, 1
Network 58
LD     V2180.5
LPS
AN     V2183.0
=      L63.7
LPP
BITIM  LD5
AENO
/D     +1000, LD5
AENO
-D     VD2190, LD5
AENO
DTI    LD5, LW0
AENO
AW>=   LW0, VW2124
O      L63.7
R      V2180.5, 1
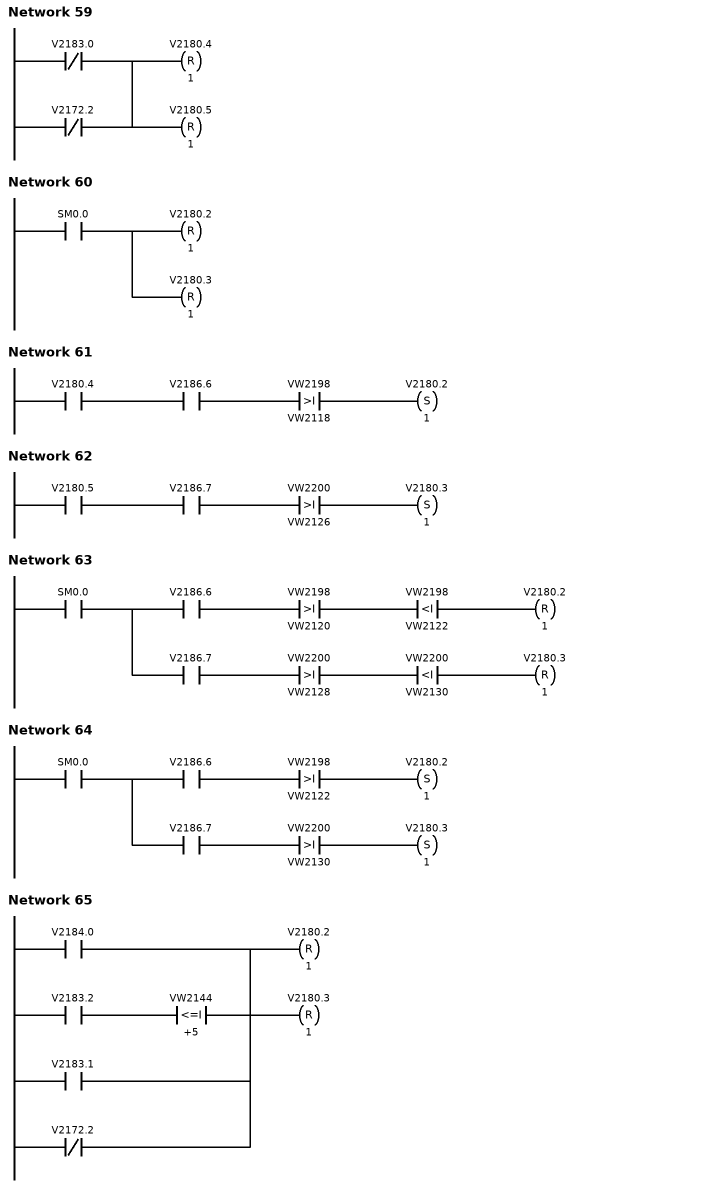
Network 59
LDN    V2183.0
ON     V2172.2
R      V2180.4, 1
R      V2180.5, 1
Network 60
LD     SM0.0
R      V2180.2, 1
R      V2180.3, 1
Network 61
LD     V2180.4
A      V2186.6
AW>    VW2198, VW2118
S      V2180.2, 1
Network 62
LD     V2180.5
A      V2186.7
AW>    VW2200, VW2126
S      V2180.3, 1
Network 63
LD     SM0.0
LPS
A      V2186.6
AW>    VW2198, VW2120
AW<    VW2198, VW2122
R      V2180.2, 1
LPP
A      V2186.7
AW>    VW2200, VW2128
AW<    VW2200, VW2130
R      V2180.3, 1
Network 64
LD     SM0.0
LPS
A      V2186.6
AW>    VW2198, VW2122
S      V2180.2, 1
LPP
A      V2186.7
AW>    VW2200, VW2130
S      V2180.3, 1
Network 65
LD     V2184.0
LD     V2183.2
AW<=   VW2144, +5
OLD
O      V2183.1
ON     V2172.2
R      V2180.2, 1
R      V2180.3, 1
END_SUBROUTINE_BLOCK

SUBROUTINE_BLOCK DATA_snd:SBR1
TITLE=
BEGIN
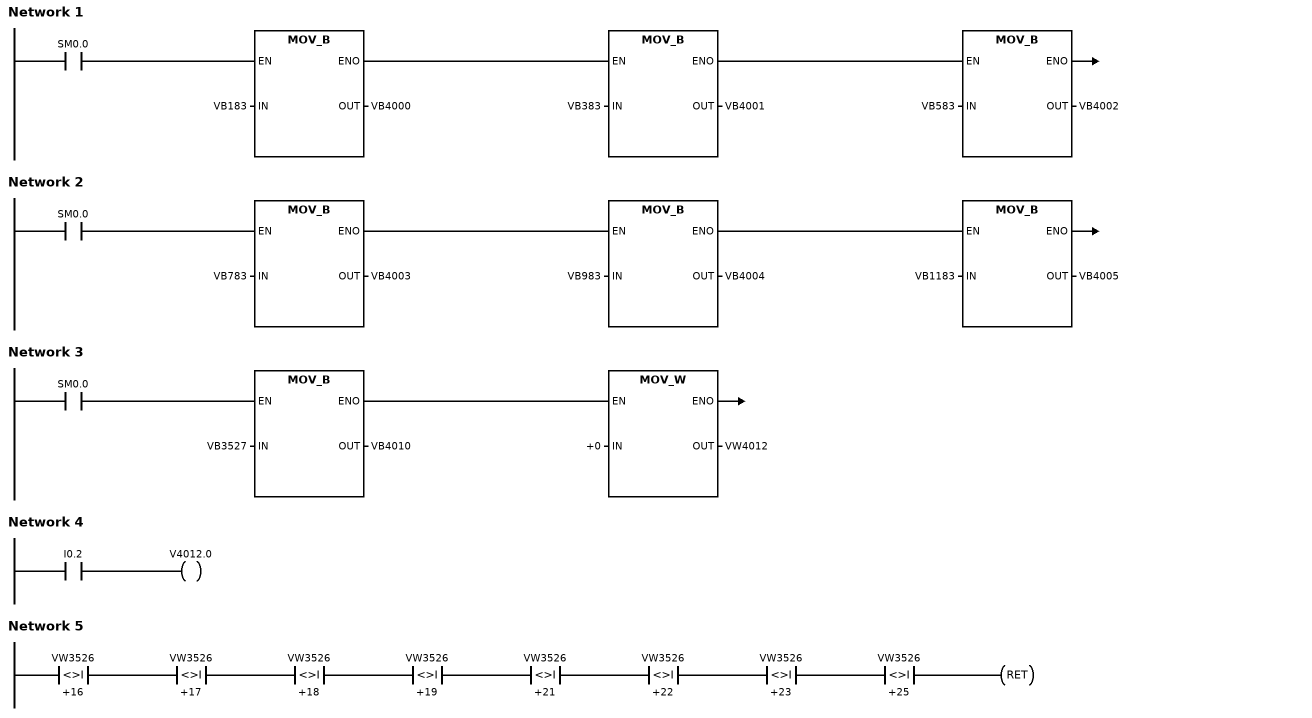
Network 1
LD     SM0.0
MOVB   VB183, VB4000
AENO
MOVB   VB383, VB4001
AENO
MOVB   VB583, VB4002
Network 2
LD     SM0.0
MOVB   VB783, VB4003
AENO
MOVB   VB983, VB4004
AENO
MOVB   VB1183, VB4005
Network 3
LD     SM0.0
MOVB   VB3527, VB4010
AENO
MOVW   +0, VW4012
Network 4
LD     I0.2
=      V4012.0
Network 5
LDW<>  VW3526, +16
AW<>   VW3526, +17
AW<>   VW3526, +18
AW<>   VW3526, +19
AW<>   VW3526, +21
AW<>   VW3526, +22
AW<>   VW3526, +23
AW<>   VW3526, +25
CRET
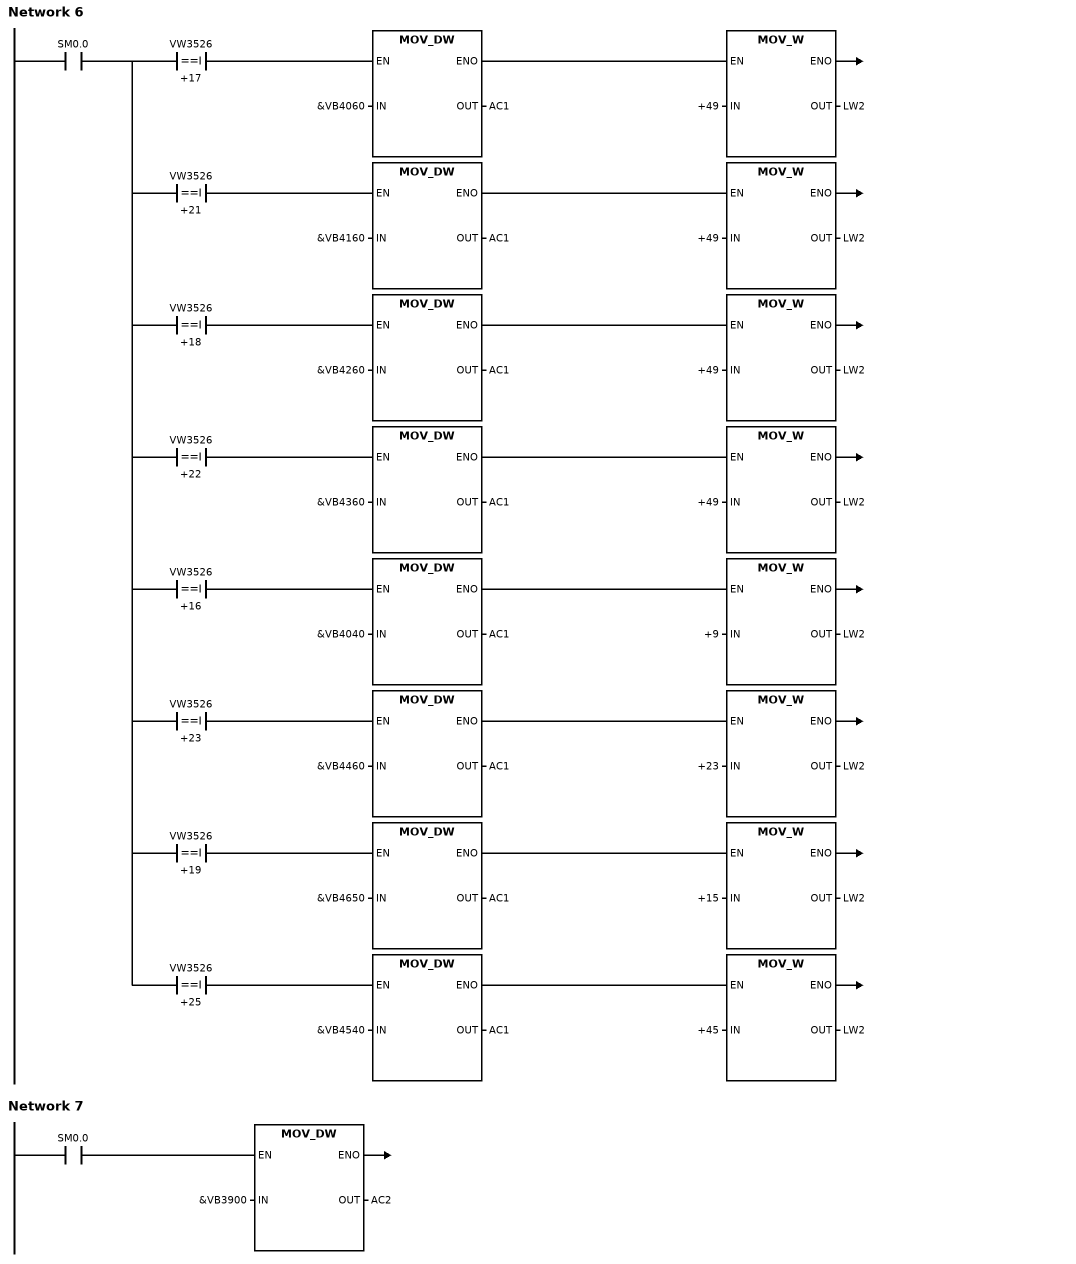
Network 6
LD     SM0.0
LPS
AW=    VW3526, +17
MOVD   &VB4060, AC1
AENO
MOVW   +49, LW2
LRD
AW=    VW3526, +21
MOVD   &VB4160, AC1
AENO
MOVW   +49, LW2
LRD
AW=    VW3526, +18
MOVD   &VB4260, AC1
AENO
MOVW   +49, LW2
LRD
AW=    VW3526, +22
MOVD   &VB4360, AC1
AENO
MOVW   +49, LW2
LRD
AW=    VW3526, +16
MOVD   &VB4040, AC1
AENO
MOVW   +9, LW2
LRD
AW=    VW3526, +23
MOVD   &VB4460, AC1
AENO
MOVW   +23, LW2
LRD
AW=    VW3526, +19
MOVD   &VB4650, AC1
AENO
MOVW   +15, LW2
LPP
AW=    VW3526, +25
MOVD   &VB4540, AC1
AENO
MOVW   +45, LW2
Network 7
LD     SM0.0
MOVD   &VB3900, AC2
